# EPICS alarm handler configuration: alh_files/mgnt_bsyA_bend.alhConfig
GROUP NULL BEND:BSYA:MG01
   $COMMAND edm -x -eolc -noedit mgnt_bsy0_bend.edl
$ALIAS BEND
$GUIDANCE
BSYA BEND
   Group Name: BEND:BSYA:MG01
   Summary PV:  BEND:BSYA:MG01:STATSUMY
$END

GROUP BEND:BSYA:MG01  BEND:BSYA:975
   $COMMAND edm -x -eolc -noedit -m "DEV=BEND:BSYA:975,PDEV=PSC:BSY0:MG06,DISP=epsc" mgnt_unit2.edl
CHANNEL    BEND:BSYA:975    BEND:BSYA:975:STATMSG   -----
   $FORCEPV BEND:BSYA:975:STATMSGSV -DATL 1 0
